(* CODESYS project motors_duts.library
   Author: Miroslav Kozarev
   Placeholder: Motors_DUTs
   Title: Motors_DUTs
   Version: 0.1
   Description: Miroslav-Sashev@sensata.com
   Company: Sensata Technologies Bulgaria

Project tree, tasks and I/O mapping:
  DUTs/
    data type E_MotorOperationModes
    data type E_MotorStates
    data type ST_MotorBase
*)

// DUTs/E_MotorOperationModes
{attribute 'qualified_only'}
TYPE E_MotorOperationModes :
(
	MODE_POSITIONING 		:= 0,
	MODE_VELOCITY			:= 1
) UDINT;
END_TYPE

// DUTs/E_MotorStates
{attribute 'qualified_only'}
TYPE E_MotorStates :
(
	MOTORSTATE_INIT,
	MOTORSTATE_ENABLE,
	MOTORSTATE_OPERATIONAL,
	MOTORSTATE_ERROR,
	MOTORSTATE_RESET,
	MOTORSTATE_MOVING,
	MOTORSTATE_MOVING_VELOCITY,
	MOTORSTATE_HOMING,
	MOTORSTATE_STOP,
	MOTORSTATE_STOP_RELEASE
) UINT;
END_TYPE

// DUTs/ST_MotorBase
TYPE ST_MotorBase :
STRUCT
	TargetPosition		: REAL;																		// The motor target position.
	TargetVelocity		: REAL;																		// The motor target velocity.
	TargetAcceleration	: REAL;																		// The motor target acceleration.
	TargetPrecision		: REAL;																		// The motor target deceleration.
	DoStop				: BOOL;																		// Use to stop the motor.
	DoEnable			: BOOL;																		// Use to enable the motor.
	DoReset				: BOOL;																		// Use to reset the motor state - if in error - reset it, else reset the motor to waiting for enable.
	DoHome				: BOOL;																		// Use to trigger encoder refference.
	DoMove				: BOOL;																		// Use to start a movement based on the passed target data.
	
	CurrentPosition		: LREAL;												                    // The current position of the motor.
	CurrentVelocity		: LREAL;																	// The current velocity of the motor.
	CurrentAcceleration	: LREAL;																	// The current acceleration of the motor.
	Enabled				: BOOL; 																	// Is the motor enabled.
	Error				: BOOL; 																	// Is the motor in an error state.
	ErrorID				: UDINT;																	// The current error state ID.
	Refferenced			: BOOL; 																	// Is the motor refferenced.
	Moving				: BOOL; 																	// Is the motor moving.
	TargetReached		: BOOL; 																	// Is the motor setpoint reached - positioning and velocity.
	OperationMode		: UDINT;																	// 0 - > Absolute position, 1 -> Velocity
END_STRUCT
END_TYPE
